TYPE st_NeedleAction :
STRUCT
	Clip				: E_NeedleClip;
	NeedlePoint			: E_NeedlePoint;
	Handshake			: ST_HandshakeBase;
END_STRUCT
END_TYPE

(* stored: Version 1.1.0.1, ProductVersion 3.1.4024.13
   DUT st_NeedleAction: Id {f85ff63c-0ca5-44a3-8d72-1fca6a074b8c} *)
